Staubli VAL3: ros_i_driver.pjx

--- ros_i_driver.pjx ---
Parameters version=s7.7.2 stackSize=5000 millimeterUnit=true
Program file=dataReceiver.pgx
Program file=dataStreamer.pgx
Program file=decTrajPt.pgx
Program file=decTrajPtFull.pgx
Program file=decodeMsgBody.pgx
Program file=decodeMsgHeader.pgx
Program file=encTrajPtAck.pgx
Program file=encTrajPtFAck.pgx
Program file=encodeAck.pgx
Program file=encodeJState.pgx
Program file=encodeJointFbk.pgx
Program file=encodeStatus.pgx
Program file=fbkStreamer.pgx
Program file=fetchStatus.pgx
Program file=initParams.pgx
Program file=motionControl.pgx
Program file=pushMotion.pgx
Program file=recvData.pgx
Program file=recvHeartbeat.pgx
Program file=recvMsgBody.pgx
Program file=recvMsgHeader.pgx
Program file=recvTrajPt.pgx
Program file=recvTrajPtFull.pgx
Program file=screenUpdate.pgx
Program file=sendAck.pgx
Program file=sendData.pgx
Program file=sendJState.pgx
Program file=sendJointFbk.pgx
Program file=sendStatus.pgx
Program file=sendTrajPtAck.pgx
Program file=sendTrajPtFAck.pgx
Program file=setupRosMsgs.pgx
Program file=start.pgx
Program file=stop.pgx
Data file=ros_i_driver.dtx
Library alias=libMoveBuffer path=Disk://MotionQueue/MotionQueue.pjx autoload=true password=
Library alias=libTrajPtBuffer path=Disk://TrajectoryQueue/TrajectoryQueue.pjx autoload=true password=
Type name=RosSimpleMsg path=Disk://RosSimpleMsg/RosSimpleMsg.pjx
Type name=RobotStatusMsg path=Disk://RobotStatusMsg/RobotStatusMsg.pjx
Type name=JointStateMsg path=Disk://JointStateMsg/JointStateMsg.pjx
Type name=JointTrajPtMsg path=Disk://JointTrajPtMsg/JointTrajPtMsg.pjx
Type name=JointTrajPtFMsg path=Disk://JointTrajPtFMsg/JointTrajPtFMsg.pjx
Type name=JointFbkMsg path=Disk://JointFbkMsg/JointFbkMsg.pjx
Type name=MotionBuffer path=Disk://MotionBuffer/MotionBuffer.pjx

--- ros_i_driver.dtx ---
public bool bFbkOverrun
public bool bMotionOverrun
public jointRx jCurrPose
public num nCounter
public num nFbkPeriod = 0.032
public num nLengthB[4]
num nMotionPeriod = 0.012
public num nPosVelAccB[120]
public num nRobotIdB[4]
public num nTimeB[4]
public num nValidFieldsB[4] = 2
public sio siTcpIpFbk = {link=Socket\Feedback}
public sio siTcpIpMotion = {link=Socket\Motion}
public string sStreamTaskName = "publisher"
public string sMotionTaskName
public num nMsgTypeB[4]
public num nReplyCodeB[4]
public bool bSendData
public num nDeg2Rad
public RosSimpleMsg rosGenericMsg
  [0]
    Header header
      [0]
        num nMsgType
        num nCommType
        num nReplyCode
        num nData[12]
    Prefix prefix
      [0]
        num nLength
        num nData[4]
public bool bValidMsgHeader
public bool bValidMsgBody
public bool bValidMotion
public jointRx jDesiredPose
public tool tTool = {fatherId=flange[0], ioLink=valve1}
public num nRad2Deg
public string sTrajPtTaskName
public bool bTrajPtOverrun
public RobotStatusMsg rosStatusMsg
  [0]
    Body body
      [0]
        num nData[28]
    Header header
      [0]
        num nMsgType
        num nCommType
        num nReplyCode
        num nData[12]
    Prefix prefix
      [0]
        num nLength
        num nData[4]
    RobotStatus robotStatus
      [0]
        num nDrivesPowered
        num nEStopped
        num nErrorCode
        num nInError
        num nInMotion
        num nMode
        num nMotionPossible
public JointStateMsg rosJointMsg
  [0]
    Header header
      [0]
        num nMsgType
        num nCommType
        num nReplyCode
        num nData[12]
    Body body
      [0]
        num nData[44]
    JointState jointState
      [0]
        num nSeq
        num nJoints[10]
    Prefix prefix
      [0]
        num nLength
        num nData[4]
public JointTrajPtMsg rosTrajPtMsg
  [0]
    Header header
      [0]
        num nMsgType
        num nCommType
        num nReplyCode
        num nData[12]
    JointTrajPt jointTrajPt
      [0]
        num nSeq
        num nJoints[10]
        num nVelocity
        num nDuration
    Prefix prefix
      [0]
        num nLength
        num nData[4]
    Body body
      [0]
        num nData[64]
public bool bRecvData
public JointTrajPtFMsg rosTrajPtFMsg
  [0]
    Header header
      [0]
        num nMsgType
        num nCommType
        num nReplyCode
        num nData[12]
    Prefix prefix
      [0]
        num nLength
        num nData[4]
    JointTrajPtFull jointTrajPtFull
      [0]
        num nRobotId
        num nSeq
        num nValidFields
        num nTime
        num nPositions[10]
        num nVelocities[10]
        num nAccelerations[10]
    Body body
      [0]
        num nData[136]
public JointFbkMsg rosJointFbkMsg
  [0]
    Header header
      [0]
        num nMsgType
        num nCommType
        num nReplyCode
        num nData[12]
    Prefix prefix
      [0]
        num nLength
        num nData[4]
    JointFeedback jointFeedback
      [0]
        num nRobotId
        num nValidFields
        num nTime
        num nPositions[10]
        num nVelocities[10]
        num nAccelerations[10]
    Body body
      [0]
        num nData[132]
public JointTrajPtFMsg rosTrajPtFAck
  [0]
    Header header
      [0]
        num nMsgType
        num nCommType
        num nReplyCode
        num nData[12]
    Prefix prefix
      [0]
        num nLength
        num nData[4]
    JointTrajPtFull jointTrajPtFull
      [0]
        num nRobotId
        num nSeq
        num nValidFields
        num nTime
        num nPositions[10]
        num nVelocities[10]
        num nAccelerations[10]
    Body body
      [0]
        num nData[136]
public bool bMsgDecoded
public bool bHeaderDecoded
public JointTrajPtMsg rosTrajPtAck
  [0]
    Header header
      [0]
        num nMsgType
        num nCommType
        num nReplyCode
        num nData[12]
    JointTrajPt jointTrajPt
      [0]
        num nSeq
        num nJoints[10]
        num nVelocity
        num nDuration
    Prefix prefix
      [0]
        num nLength
        num nData[4]
    Body body
      [0]
        num nData[64]
public bool bScreenOverrun
public string sScreenTaskName
public num nScreenUpdate
public num nTrajReception
public MotionBuffer mTrajPt
  [0]
    mdesc mVelAcc = {leave=0, reach=0}
    num nDuration
    num nSequence
    jointRx jJointRx
public num nDataIn
public num nDataOut
public num nDebugStatus
public screen scDebug
public screen scMonitor
public string sHtbtTaskName
public bool bCheckHeartbeat
public num nCommTypeB[4]
public num nBytesSent

--- start.pgx ---
program start()
begin
  // feedback task will run every 32 ms (approx. 31 Hz)
  //nFbkPeriod=0.032
  //nFbkPeriod = 0.05
  nFbkPeriod = 1.0

  // motion task will run every 12 ms (approx. 83 Hz)
  //nMotionPeriod=0.012
  nMotionPeriod = 0.05

  nTrajReception = 0.05
  nScreenUpdate = 1.0

  nDeg2Rad = 3.14159265359 / 180.0
  nRad2Deg = 180.0 / 3.14159265359

  sStreamTaskName = "streamerTask"
  sTrajPtTaskName = "trajPtTask"
  sMotionTaskName = "motionTask"
  sScreenTaskName = "screenTask"
  sHtbtTaskName = "htbtTask"

  // initialise TCP/IP parameters
  call initParams()
  // setup prefix and header of ROS messages
  call setupRosMsgs()

  // socket connections: initially disconnected
  nDataIn = 0
  nDataOut = 0

  // flags to control tasks: should start sending/receiving
  bSendData = true
  bRecvData = true
  bCheckHeartbeat = true

  nPtsPopped = 0
  nMovePts = 0

  // debug status
  nDebugStatus = 0

  // ensure motion buffer is empty
  call libTrajPtBuffer:clear()
  call libMoveBuffer:clear()

  // before anything else, enable power (only works if robot is in remote mode)
  //enablePower()
  //if (watch(isPowered(), 5) == false)
  //  popUpMsg("Arm power could not be enabled")
  //endIf

  // create joint state and robot status streamer task to send data to industrial_robot_client
  taskCreateSync sStreamTaskName, nFbkPeriod, bFbkOverrun, dataStreamer()

  // create trajectory point task to receive data from industrial_robot_client
  taskCreateSync sTrajPtTaskName, nTrajReception, bTrajPtOverrun, dataReceiver()

  // create motion task to synchronously apply motion commands to robot
  taskCreateSync sMotionTaskName, nMotionPeriod, bMotionOverrun, motionControl()

  // create synchronous task to update screen
  taskCreateSync sScreenTaskName, nScreenUpdate, bScreenOverrun, screenUpdate()

  // create asynchronous task to receive heartbeat on port 11002
  taskCreate sHtbtTaskName, 10, recvHeartbeat()

end

--- dataReceiver.pgx ---
public program dataReceiver()
begin
  //  bValidMsgHeader = false
  //  bHeaderDecoded = false
  //  bValidMsgBody = false
  //  bValidMotion = false

  // state machine at initial state
  // 0: receive header
  // 1: decode header
  // 2: receive body
  // 3: decode body
  // 4: push motion into buffer
  // 5: send ACK
  nDataInState=0

  while (bRecvData)
    // usually for state machines a switch-case statement is a neat implementation
    // HOWEVER, at every iteration of while() this task is sequenced and only called
    // after whatever ms is was defined when created.
    // As a result, receiving one single message, pushing motion and sending ACK
    // would take 6 * task period using switch-case statement.
    // The desirable behaviour is to receive and decode a full message, push motion
    // into buffer and then send ACK to client WITHIN ONE ITERATION of while(),
    // hence the if statement sequence below
    if (nDataInState==0)
      call recvMsgHeader()
    endIf
    if (nDataInState==1)
      call decodeMsgHeader()
    endIf
    if (nDataInState==2)
      call recvMsgBody()
    endIf
    if (nDataInState==3)
      call decodeMsgBody()
    endIf
    if (nDataInState==4)
      call pushMotion()
    endIf
    if (nDataInState==5)
      call encodeAck()
      call sendAck()
    endIf

    // assert state machine is working OK
    if (nDataInState<0 or nDataInState>5)
      popUpMsg("Data reception state machine error")
    endIf

    // sequence task
    delay(0)
  endWhile

  //  while (bRecvData)
  //    // receive message prefix + header
  //    call recvMsgHeader()
  //
  //    if (bValidMsgHeader)
  //      bValidMsgHeader = false
  //      // decode appropriately
  //      call decodeMsgHeader()
  //    endIf
  //
  //    if (bHeaderDecoded)
  //      bHeaderDecoded = false
  //      // receive and decode message according to msg_type
  //      switch rosGenericMsg.header.nMsgType
  //        case 11
  //          // assume Failure by default (change within decTrajPt())
  //          rosTrajPtAck.header.nReplyCode = 2
  //          //call recvTrajPt()
  //          if (bValidMsgBody)
  //            bValidMsgBody = false
  //            //call decTrajPt()
  //            // always send ACK, with reply_code = SUCCESS or FAILURE
  //            call sendAck()
  //          endIf
  //        break
  //        case 14
  //          // assume Failure by default (change within decTrajPtFull())
  //          rosTrajPtFAck.header.nReplyCode = 2
  //          //call recvTrajPtFull()
  //          if (bValidMsgBody)
  //            bValidMsgBody = false
  //            //call decTrajPtFull()
  //            // always send ACK, with reply_code = SUCCESS or FAILURE
  //            call sendAck()
  //          endIf
  //        break
  //        default
  //          bValidMsgBody = false
  //          bValidMotion = false
  //        break
  //      endSwitch
  //    endIf
  //
  //    if (bValidMotion)
  //      call pushMotion()
  //    endIf
  //
  //    // sequence task
  //    delay(0)
  //  endWhile
end

--- dataStreamer.pgx ---
public program dataStreamer()
begin
  while (bSendData)
    // fetch current joint positions
    jCurrPose=herej()
    // encode and send ROS simple_message ID 10: joint state
    call encodeJState()
    call sendJState()

    // fetch robot status
    call fetchStatus()
    // encode and send ROS simple_message ID 13: robot status
    call encodeStatus()
    call sendStatus()
    // sequence task
    delay(0)
  endWhile
end

--- decodeMsgBody.pgx ---
public program decodeMsgBody()
  local bool l_bFlag
begin
  l_bFlag = false

  switch rosGenericMsg.header.nMsgType
    case 11
      call decTrajPt(l_bFlag)
    break
    case 14
      call decTrajPtFull(l_bFlag)
    break
    default
    break
  endSwitch

  if (l_bFlag)
    // move on to state 4: push motion into buffer
    nDataInState = 4
  else
    // error whilst decoding msg body...
    if (rosGenericMsg.header.nCommType == 2)
      switch rosGenericMsg.header.nMsgType
        case 11
          rosTrajPtAck.header.nReplyCode = 2
        break
        case 14
          rosTrajPtFAck.header.nReplyCode = 2
        break
        default
        break
      endSwitch
      // jump to state 5: sendAck()
      nDataInState = 5
    else
      // reset state machine, since no ACK is required
      nDataInState = 1
    endIf
  endIf
end

--- decodeMsgHeader.pgx ---
public program decodeMsgHeader()
  local num l_nRetVal
begin
  // decode message into generic message first
  l_nRetVal=fromBinary(rosGenericMsg.prefix.nData,4,"-4l",rosGenericMsg.prefix.nLength)
  if (l_nRetVal!=1)
    // error decoding prefix, reset state machine
    nDataInState=0
    return
  endIf
  l_nRetVal=fromBinary(rosGenericMsg.header.nData,4,"-4l",rosGenericMsg.header.nMsgType)
  if (l_nRetVal!=1)
    // error decoding header (msg type), reset state machine
    nDataInState=0
    return
  endIf
  l_nRetVal=fromBinary(rosGenericMsg.header.nData[4],4,"-4l",rosGenericMsg.header.nCommType)
  if (l_nRetVal!=1)
    // error decoding header (comm type), reset state machine
    nDataInState=0
    return
  endIf
  l_nRetVal=fromBinary(rosGenericMsg.header.nData[8],4,"-4l",rosGenericMsg.header.nReplyCode)
  if (l_nRetVal!=1)
    // error decoding header (reply code), reset state machine
    nDataInState=0
    return
  endIf

  // no errors detected whilst decoding prefix and header
  // move on to state 2: receive msg body
  nDataInState=2

  //put("length: ")
  //putln(toString("", rosGenericMsg.prefix.nLength))
  //put("msg_type: ")
  //putln(toString("", rosGenericMsg.header.nMsgType))
  //put("comm_type: ")
  //putln(toString("", rosGenericMsg.header.nCommType))
  //put("reply_code: ")
  //putln(toString("", rosGenericMsg.header.nReplyCode))
end

--- decTrajPt.pgx ---
public program decTrajPt(bool& x_bFlag (dimensions=1))
  local num l_nIndex
  local num l_nRetVal
begin
  // decode message ID 11 body (data)

  // assume failure to decode
  rosTrajPtAck.header.nReplyCode=2

  // sequence
  l_nRetVal=fromBinary(rosTrajPtMsg.body.nData,4,"-4l",rosTrajPtMsg.jointTrajPt.nSeq)
  if (l_nRetVal!=1)
    x_bFlag=false
    return
  endIf

  // joints[10]
  for l_nIndex=0 to 9 step 1
    l_nRetVal=fromBinary(rosTrajPtMsg.body.nData[(l_nIndex*4)+4],4,"4.0l",rosTrajPtMsg.jointTrajPt.nJoints[l_nIndex])
    if (l_nRetVal!=1)
      x_bFlag=false
      return
    endIf
  endFor

  // velocity
  l_nRetVal=fromBinary(rosTrajPtMsg.body.nData[44],4,"4.0l",rosTrajPtMsg.jointTrajPt.nVelocity)
  if (l_nRetVal!=1)
    x_bFlag=false
    return
  endIf

  // duration
  l_nRetVal=fromBinary(rosTrajPtMsg.body.nData[48],4,"4.0l",rosTrajPtMsg.jointTrajPt.nDuration)
  if (l_nRetVal!=1)
    x_bFlag=false
    return
  endIf

  // decoding successful
  rosTrajPtAck.header.nReplyCode=1
  rosTrajPtAck.jointTrajPt.nSeq=rosTrajPtMsg.jointTrajPt.nSeq
  x_bFlag=true
end

--- decTrajPtFull.pgx ---
public program decTrajPtFull(bool& x_bFlag)
  local num l_nRetVal
  local num l_nIndex
begin
  // decode message ID 14 body (data)

  // assume failure to decode
  rosTrajPtFAck.header.nReplyCode = 2

  // robotId
  l_nRetVal = fromBinary(rosTrajPtFMsg.body.nData, 4, "-4l", rosTrajPtFMsg.jointTrajPtFull.nRobotId)
  if (l_nRetVal != 1)
    x_bFlag = false
    return
  endIf

  // sequence
  l_nRetVal = fromBinary(rosTrajPtFMsg.body.nData, 4, "-4l", rosTrajPtFMsg.jointTrajPtFull.nSeq)
  if (l_nRetVal != 1)
    x_bFlag = false
    return
  endIf

  // valid fields
  l_nRetVal = fromBinary(rosTrajPtFMsg.body.nData, 4, "-4l", rosTrajPtFMsg.jointTrajPtFull.nValidFields)
  if (l_nRetVal != 1)
    x_bFlag = false
    return
  endIf

  // time
  l_nRetVal = fromBinary(rosTrajPtFMsg.body.nData, 4, "4.0l", rosTrajPtFMsg.jointTrajPtFull.nTime)
  if (l_nRetVal != 1)
    x_bFlag = false
    return
  endIf

  // positions[10]
  for l_nIndex = 0 to 9 step 1
    l_nRetVal = fromBinary(rosTrajPtFMsg.body.nData[(l_nIndex*4)+16], 4, "4.0l", rosTrajPtFMsg.jointTrajPtFull.nPositions[l_nIndex])
    if (l_nRetVal != 1)
      x_bFlag = false
      return
    endIf
  endFor

  // velocities[10]
  for l_nIndex = 0 to 9 step 1
    l_nRetVal = fromBinary(rosTrajPtFMsg.body.nData[(l_nIndex*4)+56], 4, "4.0l", rosTrajPtFMsg.jointTrajPtFull.nVelocities[l_nIndex])
    if (l_nRetVal != 1)
      x_bFlag = false
      return
    endIf
  endFor

  // accelerations[10]
  for l_nIndex = 0 to 9 step 1
    l_nRetVal = fromBinary(rosTrajPtFMsg.body.nData[(l_nIndex*4)+96], 4, "4.0l", rosTrajPtFMsg.jointTrajPtFull.nAccelerations[l_nIndex])
    if (l_nRetVal != 1)
      x_bFlag = false
      return
    endIf
  endFor

  // decoding successful
  rosTrajPtFAck.header.nReplyCode = 1
  rosTrajPtFAck.jointTrajPtFull.nSeq = rosTrajPtFMsg.jointTrajPtFull.nSeq
  x_bFlag = true
end

--- encodeAck.pgx ---
public program encodeAck()
begin
  switch rosGenericMsg.header.nMsgType
    case 11
      call encTrajPtAck()
    break
    case 14
      call encTrajPtFAck()
    break
    default
    break
  endSwitch
end

--- encodeJointFbk.pgx ---
public program encodeJointFbk()
  local num l_nRetVal
begin
  // encode prefix length
  //l_nRetVal=toBinary(rosMsgJointFbk.prefix.nLength, 1, "-4l", nLengthB)

  // encode header
  //l_nRetVal=toBinary(rosMsgJointFbk.header.nMsgType, 1, "-4l", nMsgTypeB)
  //l_nRetVal=toBinary(rosMsgJointFbk.header.nCommType, 1, "-4l", nCommTypeB)
  //l_nRetVal=toBinary(rosMsgJointFbk.header.nReplyCode, 1, "-4l", nReplyCodeB)

  // encode first 3 variables of body message (data)
  //l_nRetVal=toBinary(rosMsgJointFbk.body.nData, 1, "-4l", nRobotIdB)
  //l_nRetVal=toBinary(rosMsgJointFbk.body.nData[1], 1, "-4l", nValidFieldsB)
  //l_nRetVal=toBinary(rosMsgJointFbk.body.nData[2], 1, "4.0l", nTimeB)

  // assuming the remaining elements have zeros assigned by default
  //rosMsgJointFbk.body.nData[3] = jCurrPose.j1
  //rosMsgJointFbk.body.nData[4] = jCurrPose.j2
  //rosMsgJointFbk.body.nData[5] = jCurrPose.j3
  //rosMsgJointFbk.body.nData[6] = jCurrPose.j4
  //rosMsgJointFbk.body.nData[7] = jCurrPose.j5
  //rosMsgJointFbk.body.nData[8] = jCurrPose.j6

  // encode 30 values representing Positions[10], Velocities[10] and Accelerations[10]
  //l_nRetVal=toBinary(rosMsgJointFbk.body.nData[3], 30, "4.0l", nPosVelAccB)
end

--- encodeJState.pgx ---
public program encodeJState()
  local num l_nRetVal
begin
  // encode prefix length
  l_nRetVal = toBinary(rosJointMsg.prefix.nLength, 1, "-4l", rosJointMsg.prefix.nData)

  // encode header
  l_nRetVal = toBinary(rosJointMsg.header.nMsgType, 1, "-4l", rosJointMsg.header.nData)
  l_nRetVal = toBinary(rosJointMsg.header.nCommType, 1, "-4l", rosJointMsg.header.nData[4])
  l_nRetVal = toBinary(rosJointMsg.header.nReplyCode, 1, "-4l", rosJointMsg.header.nData[8])

  // encode 'sequence' variable of body message (data)
  l_nRetVal = toBinary(rosJointMsg.jointState.nSeq, 1, "-4l", rosJointMsg.body.nData)

  // assuming the remaining elements have zeros assigned by default
  rosJointMsg.jointState.nJoints[0] = jCurrPose.j1 * nDeg2Rad
  rosJointMsg.jointState.nJoints[1] = jCurrPose.j2 * nDeg2Rad
  rosJointMsg.jointState.nJoints[2] = jCurrPose.j3 * nDeg2Rad
  rosJointMsg.jointState.nJoints[3] = jCurrPose.j4 * nDeg2Rad
  rosJointMsg.jointState.nJoints[4] = jCurrPose.j5 * nDeg2Rad
  rosJointMsg.jointState.nJoints[5] = jCurrPose.j6 * nDeg2Rad

  // encode 10 values representing joints[10]
  l_nRetVal = toBinary(rosJointMsg.jointState.nJoints, 10, "4.0l", rosJointMsg.body.nData[4])
end

--- encodeStatus.pgx ---
public program encodeStatus()
  local num l_nRetVal
begin
  // encode prefix length
  l_nRetVal=toBinary(rosStatusMsg.prefix.nLength,1,"-4l",rosStatusMsg.prefix.nData)

  // encode header
  l_nRetVal=toBinary(rosStatusMsg.header.nMsgType,1,"-4l",rosStatusMsg.header.nData)
  l_nRetVal=toBinary(rosStatusMsg.header.nCommType,1,"-4l",rosStatusMsg.header.nData[4])
  l_nRetVal=toBinary(rosStatusMsg.header.nReplyCode,1,"-4l",rosStatusMsg.header.nData[8])

  // encode variables of body message (data)
  l_nRetVal=toBinary(rosStatusMsg.robotStatus.nMode,1,"-4l",rosStatusMsg.body.nData)
  l_nRetVal=toBinary(rosStatusMsg.robotStatus.nEStopped,1,"-4l",rosStatusMsg.body.nData[4])
  l_nRetVal=toBinary(rosStatusMsg.robotStatus.nDrivesPowered,1,"-4l",rosStatusMsg.body.nData[8])
  l_nRetVal=toBinary(rosStatusMsg.robotStatus.nMotionPossible,1,"-4l",rosStatusMsg.body.nData[12])
  l_nRetVal=toBinary(rosStatusMsg.robotStatus.nInError,1,"-4l",rosStatusMsg.body.nData[16])
  l_nRetVal=toBinary(rosStatusMsg.robotStatus.nInMotion,1,"-4l",rosStatusMsg.body.nData[20])
  l_nRetVal=toBinary(rosStatusMsg.robotStatus.nErrorCode,1,"-4l",rosStatusMsg.body.nData[24])
end

--- encTrajPtAck.pgx ---
public program encTrajPtAck()
  local num l_nRetVal
begin
  // encode prefix length
  l_nRetVal = toBinary(rosTrajPtAck.prefix.nLength, 1, "-4l", rosTrajPtAck.prefix.nData)

  // encode header
  l_nRetVal = toBinary(rosTrajPtAck.header.nMsgType, 1, "-4l", rosTrajPtAck.header.nData)
  l_nRetVal = toBinary(rosTrajPtAck.header.nCommType, 1, "-4l", rosTrajPtAck.header.nData[4])
  l_nRetVal = toBinary(rosTrajPtAck.header.nReplyCode, 1, "-4l", rosTrajPtAck.header.nData[8])

  // encode 'sequence' variable of body message (data)
  l_nRetVal = toBinary(rosTrajPtAck.jointTrajPt.nSeq, 1, "-4l", rosTrajPtAck.body.nData)

  // encodings below are commented out to save CPU time, since values are all zeros

  // encode 10 values representing joints[10]
  //l_nRetVal = toBinary(rosTrajPtAck.jointTrajPt.nJoints, 10, "4.0l", rosTrajPtAck.body.nData[4])

  // encode 'velocity' variable of body message (data)
  //l_nRetVal = toBinary(rosTrajPtAck.jointTrajPt.nVelocity, 1, "4.0l", rosTrajPtAck.body.nData[44])

  // encode 'duration' variable of body message (data)
  //l_nRetVal = toBinary(rosTrajPtAck.jointTrajPt.nDuration, 1, "4.0l", rosTrajPtAck.body.nData[48])
end

--- encTrajPtFAck.pgx ---
public program encTrajPtFAck()
  local num l_nRetVal
begin
  // encode prefix length
  l_nRetVal = toBinary(rosTrajPtFAck.prefix.nLength, 1, "-4l", rosTrajPtFAck.prefix.nData)

  // encode header
  l_nRetVal = toBinary(rosTrajPtFAck.header.nMsgType, 1, "-4l", rosTrajPtFAck.header.nData)
  l_nRetVal = toBinary(rosTrajPtFAck.header.nCommType, 1, "-4l", rosTrajPtFAck.header.nData[4])
  l_nRetVal = toBinary(rosTrajPtFAck.header.nReplyCode, 1, "-4l", rosTrajPtFAck.header.nData[8])

  // encodings below are commented out (apart from robotId and sequence) to save CPU time, since values are all zeros

  // encode body message (data)
  l_nRetVal = toBinary(rosTrajPtFAck.jointTrajPtFull.nRobotId, 1, "-4l", rosTrajPtFAck.body.nData)
  l_nRetVal = toBinary(rosTrajPtFAck.jointTrajPtFull.nSeq, 1, "-4l", rosTrajPtFAck.body.nData[4])
  //l_nRetVal = toBinary(rosTrajPtFAck.jointTrajPtFull.nValidFields, 1, "-4l", rosTrajPtFAck.body.nData[8])
  //l_nRetVal = toBinary(rosTrajPtFAck.jointTrajPtFull.nTime, 1, "4.0l", rosTrajPtFAck.body.nData[12])

  // encode 10 values representing positions[10]
  //l_nRetVal = toBinary(rosTrajPtFAck.jointTrajPtFull.nPositions, 10, "4.0l", rosTrajPtFAck.body.nData[16])
  // encode 10 values representing velocities[10]
  //l_nRetVal = toBinary(rosTrajPtFAck.jointTrajPtFull.nVelocities, 10, "4.0l", rosTrajPtFAck.body.nData[56])
  // encode 10 values representing accelerations[10]
  //l_nRetVal = toBinary(rosTrajPtFAck.jointTrajPtFull.nAccelerations, 10, "4.0l", rosTrajPtFAck.body.nData[96])
end

--- fbkStreamer.pgx ---
public program fbkStreamer()
begin
  //bStream = true
  call setupRosMsgs()
  //while (bStream)
  while (true)
    // fetch robot status
    //call fetchStatus()

    // encode and send ROS simple message ID 13: robot status
    //call encodeStatus()
    //call sendRosMsg(rosMsgStatus)

    // fetch current joint values
    jCurrPose=herej()

    // encode and send ROS simple_message ID 15: joint feedback
    call encodeJointFbk()
    call sendJointFbk()
    delay(0)
  endWhile
end

--- fetchStatus.pgx ---
public program fetchStatus()
begin
    // fetch robot status data

    // drives_powered
    if (isPowered() == true)
      rosStatusMsg.robotStatus.nDrivesPowered = 1
    else
      rosStatusMsg.robotStatus.nDrivesPowered = 0
    endIf

    // e-stopped
    if (esStatus() == 2)
      rosStatusMsg.robotStatus.nEStopped = 1
    else
      rosStatusMsg.robotStatus.nEStopped = 0
    endIf

    // error_code
    rosStatusMsg.robotStatus.nErrorCode = -1

    // in_error
    rosStatusMsg.robotStatus.nInError = -1

    // in_motion
    if (isSettled() == true)
      rosStatusMsg.robotStatus.nInMotion = 0
    else
      rosStatusMsg.robotStatus.nInMotion = 1
    endIf

    // mode (controller/pendant mode)
    if (workingMode() == 1 or workingMode() == 2)
      rosStatusMsg.robotStatus.nMode = 1
    elseIf (workingMode() == 3 or workingMode() == 4)
      rosStatusMsg.robotStatus.nMode = 0
    else
      rosStatusMsg.robotStatus.nMode = -1
    endIf

    // motion_possible
    rosStatusMsg.robotStatus.nMotionPossible = -1
end

--- initParams.pgx ---
public program initParams()
  local num l_nRetVal
begin
  l_nRetVal=sioCtrl(siTcpIpMotion,"timeout",2)
  if (l_nRetVal!=0)
    popUpMsg("Error while setting consumer timeout")
    //return ?
  endIf

  l_nRetVal=sioCtrl(siTcpIpFbk,"timeout",2)
  if (l_nRetVal!=0)
    popUpMsg("Error while setting producer timeout")
    //return ?
  endIf
end

--- motionControl.pgx ---
public program motionControl()
  local MotionBuffer l_mTrajPt
  local bool l_bFlag
  local MotionBuffer l_motion
  local num l_nTime
  local bool l_bStopAndClean
begin
  nMoveId = -1

  while (true)
    // check connection status, and whether to stop motion
    if (nDataIn == 1 and nDataOut == 1 and bStopNow == false)

      nMotionProgress = getMoveId()

      // process trajectory point from trajectory buffer
      if (libTrajPtBuffer:nElems > 4)
        call libTrajPtBuffer:pop(l_mTrajPt, l_bFlag)
        if (l_bFlag)
          nPtsPopped = nPtsPopped + 1
          call libMoveBuffer:push(l_mTrajPt, l_bFlag)
          if (l_bFlag == false)
            //nMovePts = nMovePts + 1
          endIf
        endIf
      endIf

      // process motion command from move buffer
      // move buffer should have elements previously interpolated
      // to ensure they are 4 ms apart
      if (libMoveBuffer:nElems > 6)
        call libMoveBuffer:pop(l_motion, l_bFlag)
        if (l_bFlag)
          nMovePts = nMovePts + 1
//          if ((nMotionProgress-nMoveId) > 0.0)
//            nMoveId = movej(l_motion.jJointRx, tTool, l_motion.mDesc)
//            waitEndMove()
//            nMotionProgress = getMoveId()
//            // if this is the last motion command, call waitEndMove()
//            // to ensure point is reached
//            if (l_motion.nSequence == -1)
//              waitEndMove()
//            endIf
//          endIf
        endIf
      endIf
    else
      // stop immediately -- resetMotion() also resets moveId
      resetMotion()
      // clear buffers
      call libTrajPtBuffer:clear()
      call libMoveBuffer:clear()
      bStopNow = false

      // debug
      nPtsPopped = 0
      nMovePts = 0
    endIf

    // sequence task
    delay(0)
  endWhile
end

--- pushMotion.pgx ---
public program pushMotion()
  local bool l_bOk
  local num l_nCounter
  local num l_nJointError
begin
  switch rosGenericMsg.header.nMsgType
    case 11
      mTrajPt.nSequence=rosTrajPtMsg.jointTrajPt.nSeq

      mTrajPt.jJointRx.j1=rosTrajPtMsg.jointTrajPt.nJoints[0]
      mTrajPt.jJointRx.j2=rosTrajPtMsg.jointTrajPt.nJoints[1]
      mTrajPt.jJointRx.j3=rosTrajPtMsg.jointTrajPt.nJoints[2]
      mTrajPt.jJointRx.j4=rosTrajPtMsg.jointTrajPt.nJoints[3]
      mTrajPt.jJointRx.j5=rosTrajPtMsg.jointTrajPt.nJoints[4]
      mTrajPt.jJointRx.j6=rosTrajPtMsg.jointTrajPt.nJoints[5]

      mTrajPt.mDesc.vel=rosTrajPtMsg.jointTrajPt.nVelocity
      mTrajPt.nDuration=rosTrajPtMsg.jointTrajPt.nDuration

    break
    case 14
      mTrajPt.nSequence=rosTrajPtFMsg.jointTrajPtFull.nSeq
      mTrajPt.nDuration=rosTrajPtFMsg.jointTrajPtFull.nTime
      mTrajPt.jJointRx.j1=rosTrajPtFMsg.jointTrajPtFull.nPositions[0]
      mTrajPt.jJointRx.j2=rosTrajPtFMsg.jointTrajPtFull.nPositions[1]
      mTrajPt.jJointRx.j3=rosTrajPtFMsg.jointTrajPtFull.nPositions[2]
      mTrajPt.jJointRx.j4=rosTrajPtFMsg.jointTrajPtFull.nPositions[3]
      mTrajPt.jJointRx.j5=rosTrajPtFMsg.jointTrajPtFull.nPositions[4]
      mTrajPt.jJointRx.j6=rosTrajPtFMsg.jointTrajPtFull.nPositions[5]

      mTrajPt.mDesc.vel=rosTrajPtFMsg.jointTrajPtFull.nVelocities[0]
      mTrajPt.mDesc.accel=rosTrajPtFMsg.jointTrajPtFull.nAccelerations[0]
      mTrajPt.mDesc.decel=mTrajPt.mDesc.accel
    break
    default
    break
  endSwitch

  if (mTrajPt.nSequence==-2)
    // set flag to stop immediately
    bStopNow=true
  else
    // only push motion into buffer if not a STOP message

    call libTrajPtBuffer:push(mTrajPt,l_bOk)
    if (l_bOk==false)
      // could not push trajectory point into buffer
      // thus ACK should flag FAILURE, but only if comm type is request
      if (rosGenericMsg.header.nCommType==2)
        switch rosGenericMsg.header.nMsgType
          case 11
            rosTrajPtAck.header.nReplyCode=2
          break
          case 14
            rosTrajPtFAck.header.nReplyCode=2
          break
          default
          break
        endSwitch
      endIf
    endIf
  endIf

  // move on to state 5: send Ack
  nDataInState=5
end

--- recvData.pgx ---
public program recvData(sio& x_sTcpSocket (dimensions=1), num& x_nData[] (dimensions=1), num& x_nConnFlag (dimensions=1), bool& x_bValidFlag (dimensions=1))
  local num l_nByte
  local num l_nBytesRecv
  local num l_nIndex
begin
  // attempt to receive data on specified socket
  l_nBytesRecv=0
  l_nIndex=0
  x_bValidFlag=false

  while (l_nBytesRecv<size(x_nData))
    l_nIndex=sioGet(x_sTcpSocket,l_nByte)
    if (l_nIndex==1)
      x_nData[l_nBytesRecv]=l_nByte
      l_nBytesRecv=l_nBytesRecv+l_nIndex
      // received a byte, set flag to indicate connection
      x_nConnFlag=1
    elseIf (l_nIndex==-1)
      // error or timeout, indicate only if connection previously established
      if (x_nConnFlag==1)
        x_nConnFlag=-1
        // close connection properly (to avoid CLOSE_WAIT)
        clearBuffer(x_sTcpSocket)
      endIf
      return
    elseIf (l_nIndex>1)
      popUpMsg("sioGet() returned > 1")
      //else
      //  popUpMsg("sioGet() returned 0")
    endIf
  endWhile
  x_bValidFlag=true
end

--- recvHeartbeat.pgx ---
public program recvHeartbeat()
  local num l_nByte
  local num l_nBytesRecv
  local num l_nHtbt
  local num l_nHtbtB[4]
  local num l_nIndex
begin
  while (bCheckHeartbeat)
    // attempt to receive heartbeat
    l_nBytesRecv=0
    l_nIndex=0
    while (l_nBytesRecv<4)
      l_nIndex=sioGet(siTcpIpFbk,l_nByte)
      if (l_nIndex==1)
        l_nHtbtB[l_nBytesRecv]=l_nByte
        l_nBytesRecv=l_nBytesRecv+l_nIndex
      elseIf (l_nIndex==-1)
        // error or timeout, indicate only if connection previously established
        if (nDataOut==1)
          nDataOut=-1
          // close connection properly (to avoid CLOSE_WAIT)
          clearBuffer(siTcpIpFbk)
        endIf
      endIf
    endWhile
    // received 4 bytes
    l_nIndex=fromBinary(l_nHtbtB,4,"-4l",l_nHtbt)
    if (l_nIndex==1)
      // confirm heartbeat value -> ensure it is connected
      if (l_nHtbt==11002)
        nDataOut=1
      endIf
    endIf
  endWhile
end

--- recvMsgBody.pgx ---
public program recvMsgBody()
  local bool l_bFlag
begin
  l_bFlag=false

  switch rosGenericMsg.header.nMsgType
    case 11
      call recvTrajPt(l_bFlag)
    break
    case 14
      call recvTrajPtFull(l_bFlag)
    break
    default
    break
  endSwitch

  if (l_bFlag)
    // move on to state 3: decode msg body
    nDataInState=3
  else
    // error whilst receiving msg body, reset state machine
    nDataInState=0
  endIf
end

--- recvMsgHeader.pgx ---
public program recvMsgHeader()
  local bool l_bFlag
begin
  // attempt to receive message prefix and header
  call recvData(siTcpIpMotion,rosGenericMsg.prefix.nData,nDataIn,l_bFlag)
  if (l_bFlag)
    call recvData(siTcpIpMotion,rosGenericMsg.header.nData,nDataIn,l_bFlag)
  endIf

  if (l_bFlag)
    // move on to state 1: decode header
    nDataInState=1
  else
    // error: reset state to 0: receive header
    nDataInState=0
  endIf


  //  // attempt to receive message header
  //  l_nBytesRecv = 0
  //  l_nIndex = 0
  //
  //  while (l_nBytesRecv < 16)
  //    l_nIndex = sioGet(siTcpIpMotion, l_nByte)
  //    if (l_nIndex == -1)
  //      if (l_nBytesRecv == 0)
  //        // 11000: client is not connected?
  //        if (nDataIn == 1)
  //          nDataIn = -1
  //        endIf
  //      else
  //        // 11000: connection lost
  //        if (nDataIn == 1)
  //          nDataIn = -1
  //        endIf
  //      endIf
  //      bValidMsgHeader = false
  //      return
  //    elseIf (l_nIndex == 1)
  //      if (l_nBytesRecv < 4)
  //        rosGenericMsg.prefix.nData[l_nBytesRecv] = l_nByte
  //      else
  //        rosGenericMsg.header.nData[l_nBytesRecv-4] = l_nByte
  //      endIf
  //      l_nBytesRecv = l_nBytesRecv + l_nIndex
  //    endIf
  //  endWhile
  //  bValidMsgHeader = true
end

--- recvTrajPt.pgx ---
public program recvTrajPt(bool& x_bFlag (dimensions=1))
begin
  // attempt to receive message ID 11 data (prefix and header are in rosGenericMsg)
  rosTrajPtMsg.prefix.nLength=rosGenericMsg.prefix.nLength
  rosTrajPtMsg.header.nMsgType=rosGenericMsg.header.nMsgType
  rosTrajPtMsg.header.nCommType=rosGenericMsg.header.nCommType
  rosTrajPtMsg.header.nReplyCode=rosGenericMsg.header.nReplyCode

  call recvData(siTcpIpMotion,rosTrajPtMsg.body.nData,nDataIn,x_bFlag)


  //  // receive message ID 11 data (prefix and header are in rosGenericMsg)
  //  l_nBytesRecv = 0
  //  l_nIndex = 0
  //
  //  rosTrajPtMsg.prefix.nLength = rosGenericMsg.prefix.nLength
  //  rosTrajPtMsg.header.nMsgType = rosGenericMsg.header.nMsgType
  //  rosTrajPtMsg.header.nCommType = rosGenericMsg.header.nCommType
  //  rosTrajPtMsg.header.nReplyCode = rosGenericMsg.header.nReplyCode
  //
  //  //while (l_nBytesRecv < (rosGenericMsg.prefix.nLength - 12))
  //  while (l_nBytesRecv < 52)
  //    l_nIndex = sioGet(siTcpIpMotion, l_nByte)
  //    if (l_nIndex == -1)
  //      if (l_nBytesRecv == 0)
  //        // 11000: client is not connected?
  //        if (nDataIn == 1)
  //          nDataIn = -1
  //        endIf
  //      else
  //        // 11000: connection lost
  //        if (nDataIn == 1)
  //          nDataIn = -1
  //        endIf
  //      endIf
  //      bValidMsgBody = false
  //      return
  //    elseIf (l_nIndex == 1)
  //      rosTrajPtMsg.body.nData[l_nBytesRecv] = l_nByte
  //      l_nBytesRecv = l_nBytesRecv + l_nIndex
  //      nDataIn = 1
  //    endIf
  //  endWhile
  //  bValidMsgBody = true
end

--- recvTrajPtFull.pgx ---
public program recvTrajPtFull(bool& x_bFlag)
begin
  // receive message ID 14 data (prefix and header are in rosGenericMsg)
  rosTrajPtFMsg.prefix.nLength = rosGenericMsg.prefix.nLength
  rosTrajPtFMsg.header.nMsgType = rosGenericMsg.header.nMsgType
  rosTrajPtFMsg.header.nCommType = rosGenericMsg.header.nCommType
  rosTrajPtFMsg.header.nReplyCode = rosGenericMsg.header.nReplyCode

  call recvData(siTcpIpMotion, rosTrajPtFMsg.body.nData, nDataIn, x_bFlag)


//  // receive message ID 14 data (prefix and header are in rosGenericMsg)
//  l_nBytesRecv = 0
//  l_nIndex = 0
//
//  rosTrajPtFMsg.prefix.nLength = rosGenericMsg.prefix.nLength
//  rosTrajPtFMsg.header.nMsgType = rosGenericMsg.header.nMsgType
//  rosTrajPtFMsg.header.nCommType = rosGenericMsg.header.nCommType
//  rosTrajPtFMsg.header.nReplyCode = rosGenericMsg.header.nReplyCode
//
//  //while (l_nBytesRecv < (rosGenericMsg.prefix.nLength - 12))
//  while (l_nBytesRecv < 52)
//    l_nIndex = sioGet(siTcpIpMotion, l_nByte)
//    if (l_nIndex == -1)
//      if (l_nBytesRecv == 0)
//        // 11000: client is not connected?
//        if (nDataIn == 1)
//          nDataIn = -1
//        endIf
//      else
//        // 11000: connection lost
//        if (nDataIn == 1)
//          nDataIn = -1
//        endIf
//      endIf
//      bValidMsgBody = false
//      return
//    elseIf (l_nIndex == 1)
//      rosTrajPtFMsg.body.nData[l_nBytesRecv] = l_nByte
//      l_nBytesRecv = l_nBytesRecv + l_nIndex
//      nDataIn = 1
//    endIf
//  endWhile
//  bValidMsgBody = true
end

--- screenUpdate.pgx ---
public program screenUpdate()
begin
  userPage(scMonitor)
  cls(scMonitor)
  title(scMonitor, "ROS-I server")

  while (true)
    // clear screen
    cls(scMonitor)

    // update connection status on port 11000
    gotoxy(scMonitor, 0,0)
    // 11 characteres: gotoxy(12,0) to insert status
    put(scMonitor, "Port 11000:")
    gotoxy(scMonitor, 12,0)
    switch nDataIn
      case -1
        put(scMonitor, "connection lost")
      break
      case 0
        put(scMonitor, "not connected")
      break
      case 1
        put(scMonitor, "connected")
      break
      default
        put(scMonitor, "not connected")
      break
    endSwitch

    // update connection status on port 11002
    gotoxy(scMonitor, 0,1)
    // 11 characteres: gotoxy(12,1) to insert status
    put(scMonitor, "Port 11002:")
    gotoxy(scMonitor, 12,1)
    switch nDataOut
      case -1
        put(scMonitor, "connection lost")
      break
      case 0
        put(scMonitor, "not connected")
      break
      case 1
        put(scMonitor, "connected")
      break
      default
        put(scMonitor, "not connected")
      break
    endSwitch

    // update trajectory buffer size
    gotoxy(scMonitor, 0,3)
    // 18 characteres: gotoxy(19,3) to insert status
    put(scMonitor, "Trajectory buffer:")
    gotoxy(scMonitor, 19,3)
    put(scMonitor, libTrajPtBuffer:nElems)
    // also print number of points popped from buffer
    gotoxy(scMonitor, 24,3)
    put(scMonitor, nPtsPopped)
    // do the same for move buffer
    gotoxy(scMonitor, 0,4)
    put(scMonitor, "Motion buffer:")
    gotoxy(scMonitor, 19,4)
    put(scMonitor, libMoveBuffer:nElems)
    gotoxy(scMonitor, 24,4)
    put(scMonitor, nMovePts)

    // display nMoveId and nMotionProgress
    gotoxy(scMonitor, 0,6)
    put(scMonitor, "moveId:")
    gotoxy(scMonitor, 8,6)
    put(scMonitor, nMoveId)
    gotoxy(scMonitor, 13,6)
    put(scMonitor, "progress:")
    gotoxy(scMonitor, 23,6)
    put(scMonitor, nMotionProgress)

    // display heartbeat status
    gotoxy(scMonitor, 0,8)
    put(scMonitor, "Heartbeat status:")
    gotoxy(scMonitor, 18,8)
    put(scMonitor, nDataOut)

    // update debug status
    gotoxy(scMonitor, 18,10)
    switch nDebugStatus
      case 0
        put(scMonitor, "[+]")
        nDebugStatus = 1
      break
      case 1
        put(scMonitor, "[-]")
        nDebugStatus = 0
      break
      default
      break
    endSwitch

    // sequence task
    delay(0)
  endWhile
end

--- sendAck.pgx ---
public program sendAck()
begin
  switch rosGenericMsg.header.nMsgType
    case 11
      call sendTrajPtAck()
    break
    case 14
      call sendTrajPtFAck()
    break
    default
    break
  endSwitch

  // regardless of result from sending ACK
  // reset state machine to receive new messages
  nDataInState=0
end

--- sendData.pgx ---
public program sendData(sio& x_sTcpSocket (dimensions=1), num& x_nData[] (dimensions=1), num& x_nFlag (dimensions=1))
  local num l_nRetVal
begin
  // send data via socket connection...
  // but only if connection is alive, or
  // if heartbeat is not expected
  if (x_nFlag==1 or bCheckHeartbeat==false)
    l_nRetVal=sioSet(x_sTcpSocket,x_nData)
    if (l_nRetVal==-1)
      if (x_nFlag==1)
        x_nFlag=-1
      endIf
    elseIf (l_nRetVal<size(x_nData))
      popUpMsg("Error while sending data")
      x_nFlag=-1
    elseIf (bCheckHeartbeat==false)
      // once data is sent over an open connection,
      // flag it as connected...
      // however, it will never be possible to detect
      // disconnections because the status goes into
      // CLOSE_WAIT, but sioSet() keeps writing data
      // to the socket...
      x_nFlag=1
    endIf
  endIf
end

--- sendJointFbk.pgx ---
public program sendJointFbk()
  local num l_nRetVal
begin
  // send message length (prefix)
  l_nRetVal=sioSet(siTcpIpFbk,nLengthB)
  if (l_nRetVal==-1)
    putln("Client not connected")
    return
  elseIf (l_nRetVal<4)
    popUpMsg("Error while sending prefix")
  endIf

  nBytesSent=size(nLengthB)

  // send message header (msg type, comm type, reply code)
  l_nRetVal=sioSet(siTcpIpFbk,nMsgTypeB)
  if (l_nRetVal==-1)
    putln("Client disconnected")
    //bStream = false
    return
  elseIf (l_nRetVal<4)
    popUpMsg("Error while sending msg type")
  endIf

  nBytesSent=nBytesSent+size(nMsgTypeB)

  l_nRetVal=sioSet(siTcpIpFbk,nCommTypeB)
  if (l_nRetVal==-1)
    putln("Client disconnected")
    //bStream = false
    return
  elseIf (l_nRetVal<4)
    popUpMsg("Error while sending comm type")
  endIf

  nBytesSent=nBytesSent+size(nCommTypeB)

  l_nRetVal=sioSet(siTcpIpFbk,nReplyCodeB)
  if (l_nRetVal==-1)
    putln("Client disconnected")
    //bStream = false
    return
  elseIf (l_nRetVal<4)
    popUpMsg("Error while sending reply code")
  endIf

  nBytesSent=nBytesSent+size(nReplyCodeB)

  // send message body (data)
  // send robotId
  l_nRetVal=sioSet(siTcpIpFbk,nRobotIdB)
  if (l_nRetVal==-1)
    putln("client disconnected")
    //bStream = false
    return
  elseIf (l_nRetVal<4)
    popUpMsg("Error while sending robot ID")
  endIf

  nBytesSent=nBytesSent+size(nRobotIdB)

  // send validFields
  l_nRetVal=sioSet(siTcpIpFbk,nValidFieldsB)
  if (l_nRetVal==-1)
    putln("client disconnected")
    //bStream = false
    return
  elseIf (l_nRetVal<4)
    popUpMsg("Error while sending valid fields")
  endIf

  nBytesSent=nBytesSent+size(nValidFieldsB)

  // send Time
  l_nRetVal=sioSet(siTcpIpFbk,nTimeB)
  if (l_nRetVal==-1)
    putln("client disconnected")
    //bStream = false
    return
  elseIf (l_nRetVal<4)
    popUpMsg("Error while sending timestamp")
  endIf

  nBytesSent=nBytesSent+size(nTimeB)

  // send positions[], velocities[] and accelerations[]
  l_nRetVal=sioSet(siTcpIpFbk,nPosVelAccB)
  if (l_nRetVal==-1)
    putln("Client disconnected")
    //bStream = false
    return
  elseIf (l_nRetVal<size(nPosVelAccB))
    popUpMsg("Error while sending msg body")
  endIf

  nBytesSent=nBytesSent+size(nPosVelAccB)

  //put("Joint status sent: ")
  //putln(nBytesSent)
  //bStream = false
end

--- sendJState.pgx ---
public program sendJState()
  local num l_nRetVal
begin
  call sendData(siTcpIpFbk,rosJointMsg.prefix.nData,nDataOut)
  call sendData(siTcpIpFbk,rosJointMsg.header.nData,nDataOut)
  call sendData(siTcpIpFbk,rosJointMsg.body.nData,nDataOut)
end

--- sendStatus.pgx ---
public program sendStatus()
  local num l_nRetVal
begin
    call sendData(siTcpIpFbk, rosStatusMsg.prefix.nData, nDataOut)
    call sendData(siTcpIpFbk, rosStatusMsg.header.nData, nDataOut)
    call sendData(siTcpIpFbk, rosStatusMsg.body.nData, nDataOut)
end

--- sendTrajPtAck.pgx ---
public program sendTrajPtAck()
  local num l_nRetVal
begin
  // send message length (prefix)
  call sendData(siTcpIpMotion, rosTrajPtAck.prefix.nData, nDataIn)
  // send message header (msg type, comm type, reply code)
  call sendData(siTcpIpMotion, rosTrajPtAck.header.nData, nDataIn)
  call sendData(siTcpIpMotion, rosTrajPtAck.body.nData, nDataIn)


//  // send message length (prefix)
//  l_nRetVal = sioSet(siTcpIpMotion, rosTrajPtAck.prefix.nData)
//  if (l_nRetVal == -1)
//    putln("10000: not connected")
//    return
//  elseIf (l_nRetVal < 4)
//    popUpMsg("Error while sending prefix")
//  endIf
//
//  nBytesSent = size(rosTrajPtAck.prefix.nData)
//
//  // send message header (msg type, comm type, reply code)
//  l_nRetVal = sioSet(siTcpIpMotion, rosTrajPtAck.header.nData)
//  if (l_nRetVal == -1)
//    putln("10000: connection lost")
//    return
//  elseIf (l_nRetVal < 12)
//    popUpMsg("Error while sending msg header")
//  endIf
//
//  nBytesSent = nBytesSent + size(rosTrajPtAck.header.nData)
//
//  // send message body (data)
//  // reply_code can only be = 1 (Success) or = 2 (Failure)
//  if (rosTrajPtAck.header.nReplyCode == 2)
//    l_nRetVal = sioSet(siTcpIpMotion, rosTrajPtAck.body.nData)
//  elseIf (rosTrajPtAck.header.nReplyCode == 1)
//    l_nRetVal = sioSet(siTcpIpMotion, rosTrajPtMsg.body.nData)
//  endIf
//
//  if (l_nRetVal == -1)
//    putln("10000: connection lost")
//    return
//  elseIf (l_nRetVal < 52)
//    popUpMsg("Error while sending msg body")
//  endIf
//
//  nBytesSent = nBytesSent + size(rosTrajPtAck.body.nData)
end

--- sendTrajPtFAck.pgx ---
public program sendTrajPtFAck()
  local num l_nRetVal
begin
  // send message length (prefix)
  call sendData(siTcpIpMotion,rosTrajPtFAck.prefix.nData,nDataIn)
  // send message header (msg type, comm type, reply code)
  call sendData(siTcpIpMotion,rosTrajPtFAck.header.nData,nDataIn)
  call sendData(siTcpIpMotion,rosTrajPtFAck.body.nData,nDataIn)


  //  // send message length (prefix)
  //  l_nRetVal = sioSet(siTcpIpMotion, rosTrajPtFAck.prefix.nData)
  //  if (l_nRetVal == -1)
  //    putln("10000: not connected")
  //    return
  //  elseIf (l_nRetVal < 4)
  //    popUpMsg("Error while sending prefix")
  //  endIf
  //
  //  nBytesSent = size(rosTrajPtFAck.prefix.nData)
  //
  //  // send message header (msg type, comm type, reply code)
  //  l_nRetVal = sioSet(siTcpIpMotion, rosTrajPtFAck.header.nData)
  //  if (l_nRetVal == -1)
  //    putln("10000: connection lost")
  //    return
  //  elseIf (l_nRetVal < 12)
  //    popUpMsg("Error while sending msg header")
  //  endIf
  //
  //  nBytesSent = nBytesSent + size(rosTrajPtFAck.header.nData)
  //
  //  // send message body (data)
  //  // reply_code can only be = 1 (Success) or = 2 (Failure)
  //  if (rosTrajPtFAck.header.nReplyCode == 2)
  //    l_nRetVal = sioSet(siTcpIpMotion, rosTrajPtFAck.body.nData)
  //  elseIf (rosTrajPtFAck.header.nReplyCode == 1)
  //    l_nRetVal = sioSet(siTcpIpMotion, rosTrajPtFMsg.body.nData)
  //  endIf
  //
  //  if (l_nRetVal == -1)
  //    putln("10000: connection lost")
  //    return
  //  elseIf (l_nRetVal < 136)
  //    popUpMsg("Error while sending msg body")
  //  endIf
  //
  //  nBytesSent = nBytesSent + size(rosTrajPtFAck.body.nData)
end

--- setupRosMsgs.pgx ---
public program setupRosMsgs()
begin
  // Joint trajectory point message
  //rosMsgJointTraj.header.nMsgType=14
  //rosMsgJointTraj.header.nCommType=1
  //rosMsgJointTraj.header.nReplyCode=0

  // Feedback of joint position/velocity/acceleration
  // prefix length = 12 + 132 = 144
  //rosMsgJointFbk.prefix.nLength=144
  //rosMsgJointFbk.header.nMsgType=15
  //rosMsgJointFbk.header.nCommType=1
  //rosMsgJointFbk.header.nReplyCode=0

  // robot_id
  //rosMsgJointFbk.body.nData[0] = 0
  // valid_fields
  //rosMsgJointFbk.body.nData[1] = 2
  // time
  //rosMsgJointFbk.body.nData[2] = 3.2


  // Joint state message (ID 10)
  // prefix length = 12 + 44
  rosJointMsg.prefix.nLength = 56
  rosJointMsg.header.nMsgType = 10
  rosJointMsg.header.nCommType = 1
  rosJointMsg.header.nReplyCode = 0
  // sequence
  rosJointMsg.jointState.nSeq = 0



  // Trajectory point message (ID 11)
  // prefix length = 12 + 52
  rosTrajPtAck.prefix.nLength = 64
  rosTrajPtAck.header.nMsgType = 11
  rosTrajPtAck.header.nCommType = 3
  // reply: 1 = success, 2 = failure
  rosTrajPtAck.header.nReplyCode = 1
  // joints are assumed to be initiliased to zero

  // the message bellow will be filled upon reception
  rosTrajPtMsg.prefix.nLength = 64



  // Robot status message (ID 13)
  // prefix length = 12 + 28
  rosStatusMsg.prefix.nLength = 40
  rosStatusMsg.header.nMsgType = 13
  rosStatusMsg.header.nCommType = 1
  rosStatusMsg.header.nReplyCode = 0



  // Trajectory point full message (ID 14)
  // prefix length = 12 + 136
  rosTrajPtFAck.prefix.nLength = 148
  rosTrajPtFAck.header.nMsgType = 14
  rosTrajPtFAck.header.nCommType = 3
  // reply: 1 = success, 2 = failure
  rosTrajPtFAck.header.nReplyCode = 1
  // body (data) assumed to be initialised to zero

  // the message bellow will be filled upon reception
  rosTrajPtFMsg.prefix.nLength = 148



  // Joint feedback message (ID 15)
  // prefix length = 12 + 132
  rosJointFbkMsg.prefix.nLength = 144
  rosJointFbkMsg.header.nMsgType = 15
  rosJointFbkMsg.header.nCommType = 1
  rosJointFbkMsg.header.nReplyCode = 0
end

--- stop.pgx ---
program stop()
begin
  resetMotion()
  popUpMsg("Pending movement commands have been cancelled.")
  cls()
end
